ABB RAPID module: RightArmExample.mod

MODULE RightArmExample


    CONST speeddata movespeed:= v200;
    CONST robtarget home:=[[-9.58,-182.61,198.63],[0.0660107,-0.842421,-0.111215,-0.523069],[0,0,0,4],[-101.964,9E+9,9E+9,9E+9,9E+9,9E+9]];
    CONST robtarget cup:=[[303.05,-355.37,96.37],[0.116431,-0.991183,-0.0563017,0.028824],[1,-1,2,4],[-101.964,9E+9,9E+9,9E+9,9E+9,9E+9]];

    PROC main()


    ENDPROC
ENDMODULE
